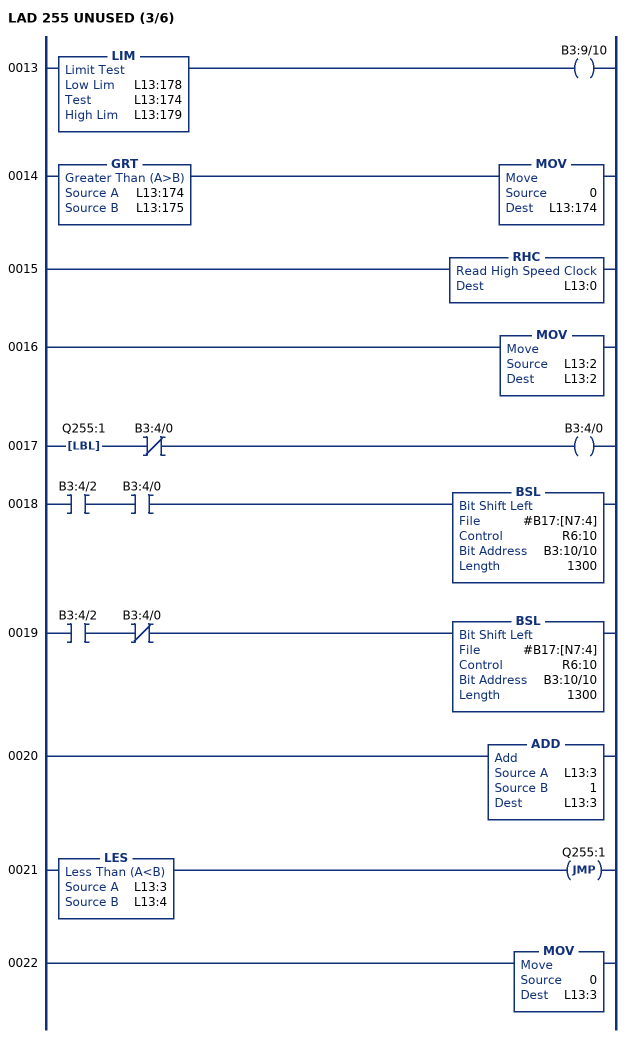
% Rung: 13 %
SOR LIM L13:178 L13:174 L13:179 OTE B3:9/10 EOR
% Rung: 14 %
SOR GRT L13:174 L13:175 MOV 0 L13:174 EOR
% Rung: 15 %
SOR RHC L13:0 EOR
% Rung: 16 %
SOR MOV L13:2 L13:2 EOR
% Rung: 17 %
SOR LBL Q255:1 XIO B3:4/0 OTE B3:4/0 EOR
% Rung: 18 %
SOR XIC B3:4/2 XIC B3:4/0 BSL #B17:[N7:4] R6:10 B3:10/10 1300 EOR
% Rung: 19 %
SOR XIC B3:4/2 XIO B3:4/0 BSL #B17:[N7:4] R6:10 B3:10/10 1300 EOR
% Rung: 20 %
SOR ADD L13:3 1 L13:3 EOR
% Rung: 21 %
SOR LES L13:3 L13:4 JMP Q255:1 EOR
% Rung: 22 %
SOR MOV 0 L13:3 EOR

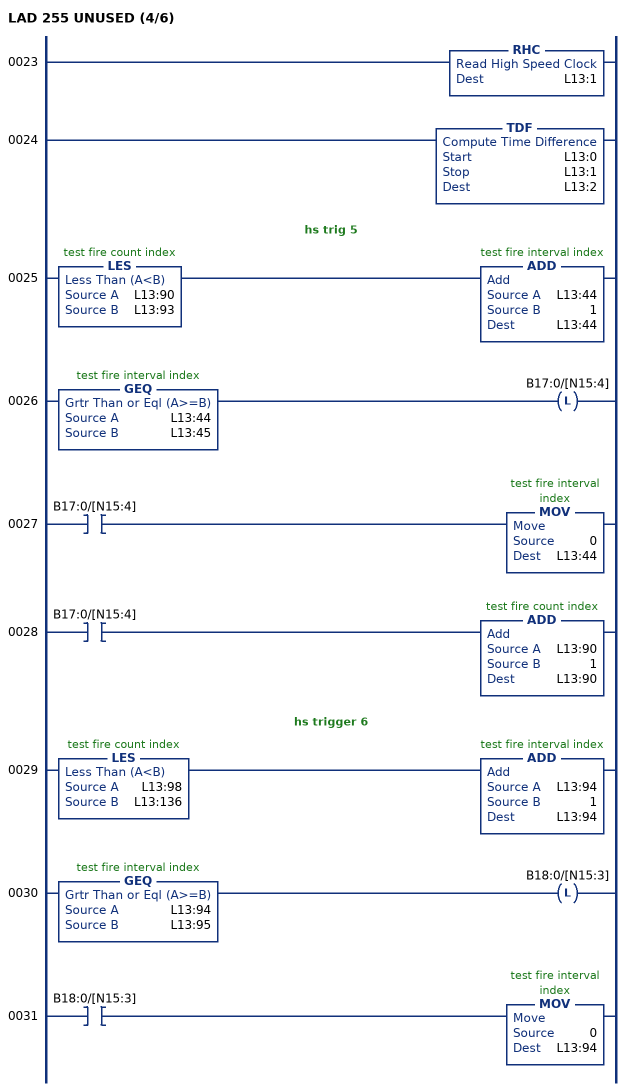
% Rung: 23 %
SOR RHC L13:1 EOR
% Rung: 24 %
SOR TDF L13:0 L13:1 L13:2 EOR
% Rung: 25 %
% TITLE: hs trig 5 %
SOR LES L13:90 L13:93 ADD L13:44 1 L13:44 EOR
%   L13:90  "test fire count index" %
%   L13:93  "test fire count" %
%   L13:44  "test fire interval index" %
% Rung: 26 %
SOR GEQ L13:44 L13:45 OTL B17:0/[N15:4] EOR
%   L13:44  "test fire interval index" %
%   L13:45  "test fire interval" %
%   B17:0  GOOD1 %
%   N15:4  INS_5_TRIG_LOC %
% Rung: 27 %
SOR XIC B17:0/[N15:4] MOV 0 L13:44 EOR
%   B17:0  GOOD1 %
%   N15:4  INS_5_TRIG_LOC %
%   L13:44  "test fire interval index" %
% Rung: 28 %
SOR XIC B17:0/[N15:4] ADD L13:90 1 L13:90 EOR
%   B17:0  GOOD1 %
%   N15:4  INS_5_TRIG_LOC %
%   L13:90  "test fire count index" %
% Rung: 29 %
% TITLE: hs trigger 6 %
SOR LES L13:98 L13:136 ADD L13:94 1 L13:94 EOR
%   L13:98  "test fire count index" %
%   L13:136  "test fire count" %
%   L13:94  "test fire interval index" %
% Rung: 30 %
SOR GEQ L13:94 L13:95 OTL B18:0/[N15:3] EOR
%   L13:94  "test fire interval index" %
%   L13:95  "test fire interval" %
%   B18:0  GOOD2 %
%   N15:3  INS_6_TRIG_LOC %
% Rung: 31 %
SOR XIC B18:0/[N15:3] MOV 0 L13:94 EOR
%   B18:0  GOOD2 %
%   N15:3  INS_6_TRIG_LOC %
%   L13:94  "test fire interval index" %

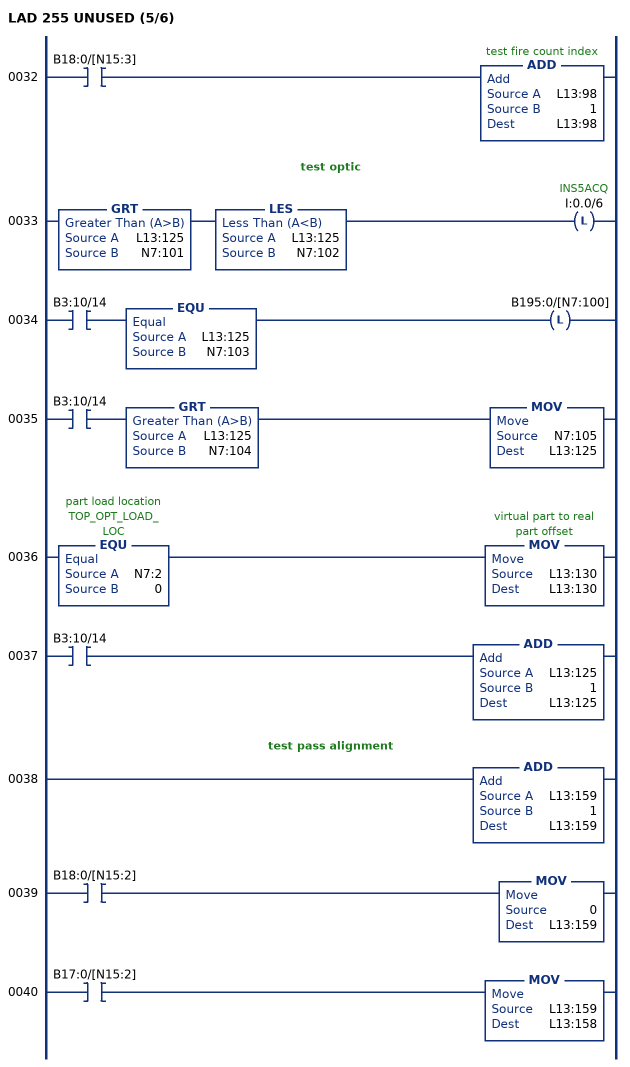
% Rung: 32 %
SOR XIC B18:0/[N15:3] ADD L13:98 1 L13:98 EOR
%   B18:0  GOOD2 %
%   N15:3  INS_6_TRIG_LOC %
%   L13:98  "test fire count index" %
% Rung: 33 %
% TITLE: test optic %
SOR GRT L13:125 N7:101 LES L13:125 N7:102 OTL I:0.0/6 EOR
%   I:0.0/6  INS5ACQ %
% Rung: 34 %
SOR XIC B3:10/14 EQU L13:125 N7:103 OTL B195:0/[N7:100] EOR
%   B195:0  TOP_NG %
% Rung: 35 %
SOR XIC B3:10/14 GRT L13:125 N7:104 MOV N7:105 L13:125 EOR
% Rung: 36 %
SOR EQU N7:2 0 MOV L13:130 L13:130 EOR
%   N7:2  TOP_OPT_LOAD_LOC  "part load location" %
%   L13:130  "virtual part to real part offset" %
% Rung: 37 %
SOR XIC B3:10/14 ADD L13:125 1 L13:125 EOR
% Rung: 38 %
% TITLE: test pass alignment %
SOR ADD L13:159 1 L13:159 EOR
% Rung: 39 %
SOR XIC B18:0/[N15:2] MOV 0 L13:159 EOR
%   B18:0  GOOD2 %
%   N15:2  BLOW_PT %
% Rung: 40 %
SOR XIC B17:0/[N15:2] MOV L13:159 L13:158 EOR
%   B17:0  GOOD1 %
%   N15:2  BLOW_PT %

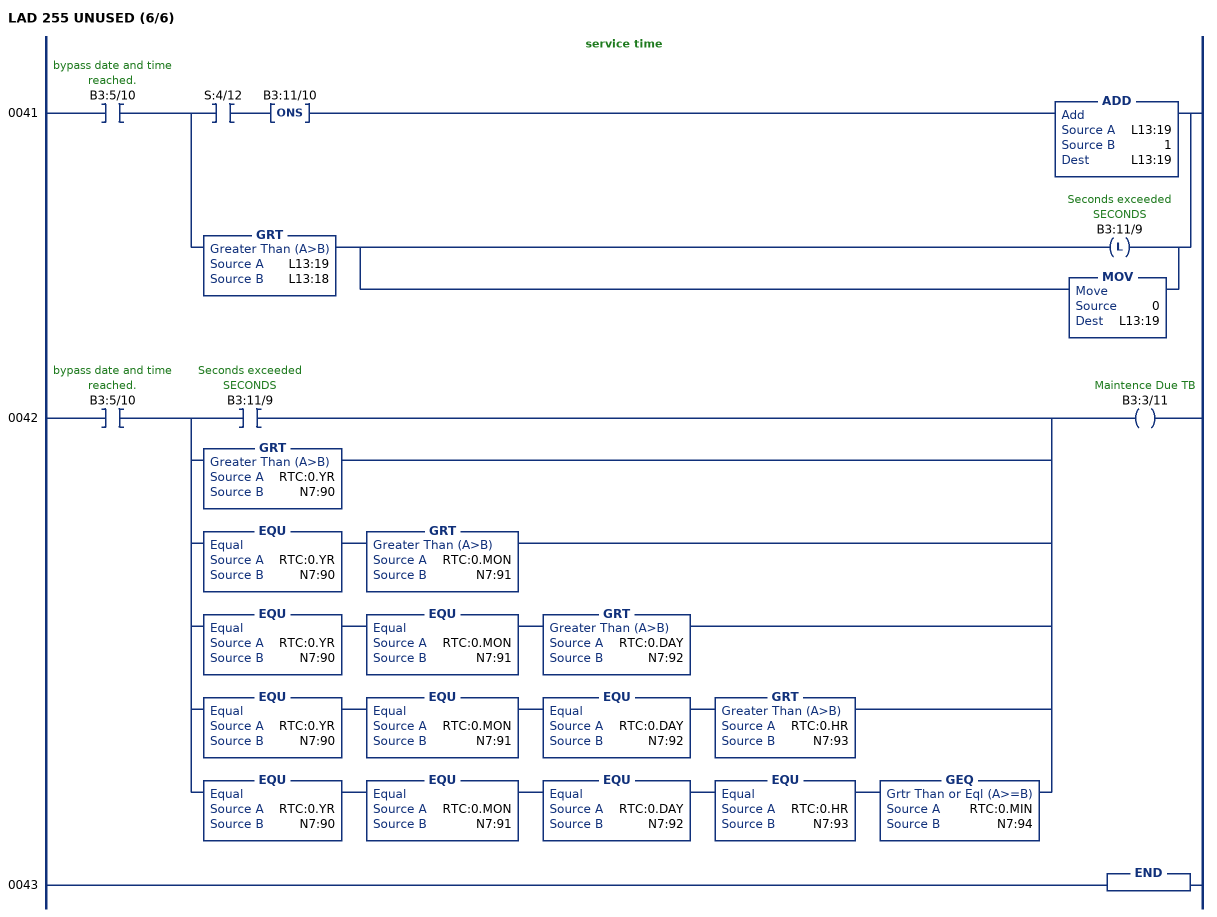
% Rung: 41 %
% TITLE: service time %
SOR XIC B3:5/10 BST XIC S:4/12 ONS B3:11/10 ADD L13:19 1 L13:19 NXB GRT L13:19 L13:18 BST OTL B3:11/9 NXB MOV 0 L13:19 BND BND EOR
%   B3:5/10  "bypass date and time reached." %
%   L13:18  MAX %
%   B3:11/9  SECONDS  "Seconds exceeded" %
% Rung: 42 %
SOR XIC B3:5/10 BST XIC B3:11/9 NXB GRT RTC:0.YR N7:90 NXB EQU RTC:0.YR N7:90 GRT RTC:0.MON N7:91 NXB EQU RTC:0.YR N7:90 EQU RTC:0.MON N7:91 GRT RTC:0.DAY N7:92 NXB EQU RTC:0.YR N7:90 EQU RTC:0.MON N7:91 EQU RTC:0.DAY N7:92 GRT RTC:0.HR N7:93 NXB EQU RTC:0.YR N7:90 EQU RTC:0.MON N7:91 EQU RTC:0.DAY N7:92 EQU RTC:0.HR N7:93 GEQ RTC:0.MIN N7:94 BND OTE B3:3/11 EOR
%   B3:5/10  "bypass date and time reached." %
%   B3:11/9  SECONDS  "Seconds exceeded" %
%   N7:90  RTC %
%   B3:3/11  TB  "Maintence Due" %
% Rung: 43 %
SOR END EOR

OTHER DOCUMENTED ADDRESSES
  B3  
  B196:0/2  ON
  B196:0/3  OFF
  B196:0/10  TOP_MOVE  "top movement detected"
  B196:1/2  DOWNTRACK_OPTIC_RUN  "Feed Bowl optic Run Signal after timing delays"
  I:0.0/0  TOP_CONV_ENC_A
  I:0.0/1  TOP_CONV_ENC_B
  I:0.0/8  INS5NG
  I:0.7  "Air Presure Sensor Input Signal"
  L42:0/2  "box full read (unused)"
  L42:1/1  "ps stop write (unused)"
  L199:9  "ones"
  L199:10  "billions"
  N15:9  FEED_WHEEL_STOP_TIME
  N197:7  "down track on delay"
  N197:8  "down track off delay"
  O:0.0/0  "spare"
  O:0.0/9  "spare"
  O:0.0/10  "spare"
  O:0.0/11  "spare"
  PFILE:6  "check for part jams"
  PFILE:10  "Bottom belt HSC"
  PFILE:12  "Top belt HSC"
  Q2:55  END_OF_MAIN
  U:6  "feed"
  U:217  "test trigger"

COMMENTS NOT ATTACHED TO A CURRENT RUNG
  F8:13: *************************
    Loads Side Camera Passing data into a bit shift
    *************************
    
    loads passing data bit into passing data bit shift register at the part present cl.
  I:0.0/8: special rung for testing. This rung can simulate a pass signal. It will not be timed correctly.
  B23:0/0: Yet another bit shift load with data in the part position indicating that there was a bottom system part pass as well as a top system part present at this location.
    
    verified works w/bypassed 071910 and unbypassed 072010
  C5:4: tempory counting to verify pass part count with boxing part count.
  B22:0/0: ***********************
     Bottom Part Syncronizing Logic
    ***********************
    
    This is the point at the bottom of the top conveyor where the part jumps from the bottom conveyor.  This system will then track the part through the top system to the point of the laser optic in order to verify that the part in question has passed the bottom inspection.  I believe that we NEED to include FAILING inspections to eliminate the possibility of a out of position part from passing. LW 072010
  T20:2.ACC: This rung is starting a timer that should be activated directly before the laser optic part presense sensor on the top conveyer and should cause the top optic to be ignored if the bottom camera system didn't pass. however other arrangements must be made if the bottom camera isn't going to be used as is the case with a nut inspection.
  T20:2: The timer used to verify that the part that triggered the top laser optic has passed the bottom camer. needs to be count
  N17:8: ****************************************************************************************************************
    I can not find anywhere in the program where the "Test Spacing From Pickup to Trigger is activated indicating to me that this entire function must not be doing anything in this program at this time.
    ****************************************************************************************************************
  B11:0/0: load part present bit shit with one shot data from the part present sensor
  B3:7/9: ************************************
     The next 3 rungs appear to do nothing
    ***********************************
  B9:0/[N7:47]: Remove any part present signals outside of expected location
  B9:0/[N7:50]: Remove any part present signals outside of expected location
  F19:0: Counter inside of a high speed counter interrupt counts the number of Bit Shifts that need to be processed in order to move the logic with the parts on the conveyor.
  F8:14: **************
    Bottom Top Camera Trigger
    *************
    
    Trigger Bottom Top Camera
  N10:4: test if boxing is connected
  B3:11/3: After initial delay allow blow two start functioning
  RUNG000150-000011: trigger count
  RUNG000150-000012: wipe stored part data if acq time expires
  RUNG000150-000013: clear data for aquire time expired
  RUNG000150-000014: clear data for time
  RUNG000150-000016: wiped count
  RUNG000150-000018: pass, fail and acquire inputs
  RUNG000150-000025: pass code / Set pass bit in Bit Shift
    captures result position and processing time
    Unlatch pass bit
  RUNG000150-000032: pass count
  RUNG000150-000035: fail count
  RUNG000150-000038: acquire code
  RUNG000150-000039: Grab trigger/acquire position
    Grab acquire time
  RUNG000150-000041: transfer tracked part positon from trigger/acquire to the acquire/result
    capture acquire time
    reset process time
  L14:8: on when ok for run
  L14:3: off when ok to run
  L14:2: off when ok to run
  L14:5: on when ok to run, rear off turns both off
  L13:165: maximum q i1
  N7:76: removed relieance on trigger signal
  N197:20/0: Passes deformed head blowoff command to TOP PLC where solenoid output is located.
  L13:162: maximum q
  L13:163: maximum average q
  B3:10/1: prevents momentary signals from box present sensor from tripping the logic for box not present
    
    This is in responce to a problem created by the sensor occasionally turning on as if no box was in its path when there is a box present.
  B3:6/2: IF PROCESSING FAULT OCURES AT COUNTER SENSOR; CLEAR THE BELT OF PASSING DATA
  L14:23: ****************  nEEDS fIXING  **********************
  L14:36: ****************  nEEDS fIXING  **********************
  RUNG000010-000014: ****
                      Zeros out the non passing part count when one passes
    ****
  RUNG000010-000018: Remove any part present signals outside of expected location
  T4:26: Check for buffer reset
  RUNG000125-000014: clear data for time
  RUNG000125-000013: clear data for aquire time expired
  RUNG000125-000012: wipe stored part data if acq time expires
  RUNG000125-000011: trigger count
  RUNG000125-000029: Set pass bit in Bit Shift
    captures result position and processing time
    Unlatch pass bit
  RUNG000125-000027: transfer tracked part positon from trigger/acquire to the acquire/result
    capture acquire time
    reset process time
  RUNG000125-000026: Grab trigger/acquire position
    Grab acquire time
  RUNG000125-000025: pass code / Set pass bit in Bit Shift
    captures result position and processing time
    Unlatch pass bit
  RUNG000125-000018: pass, fail and acquire inputs
  RUNG000125-000016: wiped count

REVISION NOTES
  13: updated count reset
  14: added io moduals
  15: multiple steps toward new hmi integration
  21: test

DATA TABLE (non-zero values as saved)
DATA B3
% B3:0 % 0X0120 0X0060 0X02C9 0XA000 0XA92E 0X2061 0X08A2 0X2AA6 0X2130 0X6104
% B3:10 % 0X8082 0X084C 0X2000 0X0000 0X0000 0X0000 0X0000 0X0000 0X0000 0X0000
DATA T4
% .PRE .ACC %
% T4:0 % 555 468
% T4:1 % 222 21
% T4:2 % 600 0
% T4:3 % 1000 1000
% T4:4 % 1 0
% T4:5 % 666 0
% T4:6 % 30 0
% T4:7 % 250 0
% T4:8 % 250 0
% T4:9 % 50 24
% T4:10 % 200 200
% T4:11 % 666 0
% T4:12 % 40 80
% T4:13 % 6 3
% T4:14 % 250 0
% T4:15 % 222 119
% T4:16 % 222 122
% T4:17 % 100 75
% T4:18 % 30 0
% T4:19 % 300 0
% T4:20 % 200 0
% T4:21 % 200 0
% T4:22 % 200 0
% T4:23 % 250 0
% T4:24 % 100 0
% T4:25 % 100 0
% T4:26 % 10 11
% T4:27 % 21 0
% T4:28 % 250 0
% T4:29 % 5000 0
% T4:30 % 50 50
% T4:31 % 20 0
% T4:32 % 69 0
DATA C5
% .PRE .ACC %
% C5:0 % 32766 0
DATA R6
% .LEN .POS %
% R6:0 % 2048 0
% R6:1 % 2048 0
% R6:2 % 3 0
% R6:3 % 3 0
% R6:4 % 1250 0
% R6:5 % 1250 0
% R6:6 % 1250 0
% R6:7 % 10 0
% R6:8 % 3 0
% R6:9 % 3 0
% R6:10 % 1300 0
% R6:11 % 1300 0
% R6:12 % 10 0
% R6:13 % 10 0
% R6:14 % 10 0
% R6:15 % 10 0
% R6:16 % 1100 0
% R6:17 % 1440 0
% R6:18 % 1440 0
% R6:19 % 10 0
DATA N7
% N7:0 % 3339 1 1168 0 0 0 49 0 1 0
% N7:10 % 48 62 1 47 1378 250 555 100 32468 96
% N7:20 % 0 73 0 0 1 10 9 1190 4096 13
% N7:30 % 50 9 800 555 222 3 1533 222 1165 222
% N7:40 % 2100 2158 10 5 2153 10 101 2050 50 1542
% N7:50 % 1552 800 10 41 0 0 1542 1552 10 41
% N7:60 % 0 0 1051 40 47 1946 1947 1944 1943 0
% N7:70 % 0 21 23 27738 32767 0 122 0 16 0
% N7:80 % 0 6 95 0 0 0 5 500 0 0
% N7:90 % 2011 4 4 12 1 0 0 0 0 1600
% N7:100 % 1003 90 110 100 175 25 0 0 0 0
DATA F8
% F8:0 % 18 206.64 23807 499 0.23807
% F8:5 % 0 0 500 1.9 2
% F8:10 % 1 0.08897486 0 101 63.26563
% F8:15 % 37.73437 4040 2 0 0
% F8:20 % 0 0.02 0 1 0
% F8:25 % 0 932781 0.222 279.6551 848597
% F8:30 % 0 170 0.03 38 852060
% F8:35 % 0 0 0 0 77
% F8:40 % 101 37.73437 0 100 1
% F8:45 % 1 2 0.21455 0 0
% F8:50 % 0 0 1 0 1
% F8:55 % 2000000 -221 0 0 0
% F8:95 % 0 0 0 492 4.92
DATA B12
% B12:0 % 0X0554 0X0000 0X0000 0X0000 0X0000 0X0000 0X0000 0X0000 0X0000 0X0000
DATA L13
% L13:0 % 308402300 308407124 4824 0 1000
% L13:5 % 0 -1901611778 100 1162124017 1162124017
% L13:10 % 492 300 78447 0 -885760695
% L13:15 % -1282263690 -2147483648 2147483647 2147483647 82058
% L13:20 % 6000000 -1295363090 0 -1144258314 2035272617
% L13:25 % 27 849 623 0 1000000000
% L13:30 % -1144259014 78452 2044398469 13 156899
% L13:35 % 678 156899 2044398469 37 2035272617
% L13:40 % -1283018330 0 19 20 0
% L13:45 % 60 700 27 0 16
% L13:50 % 0 35 666 50 3
% L13:55 % 0 1353 1297 226 226
% L13:60 % 8 10576 13 2044398343 12
% L13:65 % 650492 20 379089 1507595048 5501
% L13:70 % 1507612018 1507611965 53 0 5500
% L13:75 % -1 10 2377213 -1313930933 2377
% L13:80 % 27 -47 18250 0 999999
% L13:85 % 6475 291 44441 -1282752161 -1282751687
% L13:90 % 26616 0 0 1000 0
% L13:95 % 60 0 0 25989 488545
% L13:100 % 488093 -1282752128 -1282751656 4 3
% L13:105 % -1295599743 -1295599743 0 0 0
% L13:110 % 75 33 31 -1303967890 -1303588810
% L13:115 % -1303588792 18 9 -1303588801 5
% L13:120 % 33 10337 19 30 31
% L13:125 % 164 -1295599743 -1295599743 13 13
% L13:130 % 5 0 1 558 0
% L13:135 % 0 1000 226 12 0
% L13:140 % 0 1 12 0 20
% L13:145 % 1 34396982 35155 6 6
% L13:150 % 5 5 5 5 5
% L13:155 % 5 5 24 0 168160
% L13:160 % 3 5 4 395082 53203921
% L13:165 % 3 189116 95 13 0
% L13:170 % 55946610 0 0 1 30
% L13:175 % 300 5 5 0 10
% L13:180 % 5 6946 1000 22 1000
% L13:185 % 55 172460 60 1 720323
% L13:190 % 65 0 1 379089 379089
% L13:195 % -2370948 2370948 0 0 0
DATA F14
% F14:0 % 760.1599 200.1099 76 20 15
% F14:5 % 32766 21297.9 0 0 0
DATA N15
% N15:0 % 100 889 1945 1201 1200 134 105 100 1159 10
% N15:10 % 61 504 0 0 0 0 1172 0 0 0
DATA L16
% L16:0 % 12 40 72 0 20
% L16:5 % 250 5000 5000 182 19
% L16:10 % 1256 18 2045 6599584 98
% L16:15 % 99 0 0 0 0
DATA B17
% B17:50 % 0X0000 0X0010 0X0000 0X0000 0X0000 0X0000 0X0000 0X0000 0X0000 0X0000
DATA B18
% B18:50 % 0X0000 0X0010 0X0000 0X0000 0X0000 0X0000 0X0000 0X0000 0X0000 0X0000
% B18:60 % 0XC000 0X0000 0X0000 0X0000 0X0000 0X0000 0X0000 0X0000 0X0000 0X0000
DATA L19
% L19:0 % -1144266694 -1144265339 -1144265113 -1144263756 -1144263531
% L19:5 % -1144262174 -1144261949 -1144260596 -1144260370 -1144259014
% L19:10 % -1144258788 -1144296955 -1144296727 -1144295373 -1144295147
% L19:15 % -1144293793 -1144293568 -1144292213 -1144291988 -1144290632
% L19:20 % -1144290404 -1144289051 -1144288825 -1144287470 -1144287244
% L19:25 % -1144285888 -1144285664 -1144284312 -1144284086 -1144282731
% L19:30 % -1144282504 -1144281152 -1144280926 -1144279570 -1144279344
% L19:35 % -1144277988 -1144277763 -1144276410 -1144276184 -1144274826
% L19:40 % -1144274600 -1144273248 -1144273021 -1144271667 -1144271441
% L19:45 % -1144270087 -1144269861 -1144268503 -1144268276 -1144266921
DATA L20
% L20:0 % 2072136995 2072136995 2072136995 2072136995 2072136995
% L20:5 % 2072136995 2072136995 2072136995 2072136995 2072136995
% L20:10 % 2072136995 2072136995 2072136995 2072136995 2072136995
% L20:15 % 2072136995 2072136995 2072136995 2072136995 2072136995
% L20:20 % 2072136995 2072136995 2072136995 2072136995 2072136995
% L20:25 % 2072136995 2072136995 2072136995 2072136995 2072136995
% L20:30 % 2072136995 2072136995 2072136995 2072136995 2072136995
% L20:35 % 2072136995 2072136995 2072136995 2072136995 2072136995
% L20:40 % 2072136995 2072136995 2072136995 2072136995 2072136995
% L20:45 % 2072136995 2072136995 2072136995 2072136995 2072136995
DATA L21
% L21:0 % -1144296045 -1144294690 -1144294463 -1144293109 -1144292883
% L21:5 % -1144291527 -1144291301 -1144289948 -1144289722 -1144288365
% L21:10 % -1144288138 -1144286784 -1144286558 -1144285206 -1144284981
% L21:15 % -1144283624 -1144283398 -1144282042 -1144281817 -1144280464
% L21:20 % -1144280238 -1144278886 -1144278660 -1144277303 -1144277076
% L21:25 % -1144275718 -1144275492 -1144274137 -1144273911 -1144272559
% L21:30 % -1144272332 -1144270977 -1144270750 -1144269393 -1144269167
% L21:35 % -1144267809 -1144267584 -1144266229 -1144266003 -1144264646
% L21:40 % -1144264419 -1144263062 -1144262836 -1144261481 -1144261254
% L21:45 % -1144259899 -1144259674 -1144258314 -1144258088 -1144296272
DATA L22
% L22:0 % 2072136995 2072136995 2072136995 2072136995 2072136995
% L22:5 % 2072136995 2072136995 2072137059 2072136995 2072136995
% L22:10 % -75280985 2072136995 2072137067 2072137059 2072137523
% L22:15 % 2072137059 2072137059 2072136995 2072137059 2072136995
% L22:20 % 2072136995 -74821853 2072136995 2139245859 2072136995
% L22:25 % 2072136995 2072145779 2074242403 2073189795 -75346653
% L22:30 % 2072399203 2072136995 2072136995 2072136995 2072407459
% L22:35 % 2072669475 2072136995 2072136995 2072136995 2072136995
% L22:40 % 2072169831 2141343523 2072136995 2072136995 2074234147
% L22:45 % 2072169891 2074496803 2072247603 2074234147 2072136995
DATA L23
% L23:0 % -1304697501 -1304696943 -1304696384 -1304695825 -1304695268
% L23:5 % -1304694711 -1304694153 -1282753837 -1282753278 -1282752719
% L23:10 % -1282752161 -1304719281 -1304718723 -1304718164 -1304717606
% L23:15 % -1304717048 -1304716490 -1304715930 -1304715371 -1304714813
% L23:20 % -1304714254 -1304713694 -1304713136 -1304712578 -1304712020
% L23:25 % -1304711462 -1304710903 -1304710345 -1304709788 -1304709228
% L23:30 % -1304708671 -1304708112 -1304707554 -1304706995 -1304706437
% L23:35 % -1304705879 -1304705321 -1304704763 -1304704205 -1304703647
% L23:40 % -1304703088 -1304702530 -1304701970 -1304701411 -1304700853
% L23:45 % -1304700292 -1304699733 -1304699175 -1304698617 -1304698059
DATA L24
% L24:0 % -1295599743 -1295599743 -1295599743 -1295599743 -1295599743
% L24:5 % -1295599743 -1295599743 -1295599743 -1295599743 -1295599743
% L24:10 % -1295599743 -1295599743 -1295599743 -1295599743 -1295599743
% L24:15 % -1295599743 -1295599743 -1295599743 -1295599743 -1295599743
% L24:20 % -1295599743 -1295599743 -1295599743 -1295599743 -1295599743
% L24:25 % -1295599743 -1295599743 -1295599743 -1295599743 -1295599743
% L24:30 % -1295599743 -1295599743 -1295599743 -1295599743 -1295599743
% L24:35 % -1295599743 -1295599743 -1295599743 -1295599743 -1295599743
% L24:40 % -1295599743 -1295599743 -1295599743 -1295599743 -1295599743
% L24:45 % -1295599743 -1295599743 -1295599743 -1295599743 -1295599743
DATA L25
% L25:0 % -1282767881 -1282767655 -1282767430 -1282767205 -1282766980
% L25:5 % -1282766755 -1282766529 -1282766305 -1282766079 -1282765855
% L25:10 % -1282765628 -1282765402 -1282765177 -1282764951 -1282764727
% L25:15 % -1282764501 -1282764276 -1282764050 -1282763825 -1282763600
% L25:20 % -1282756416 -1282756192 -1282755967 -1282755743 -1282755517
% L25:25 % -1282755291 -1282755067 -1282754841 -1282754616 -1282754391
% L25:30 % -1282754165 -1282753940 -1282753715 -1282753489 -1282753264
% L25:35 % -1282753038 -1282752813 -1282752589 -1282752362 -1282752137
% L25:40 % -1282751913 -1282751687 -1282769681 -1282769457 -1282769231
% L25:45 % -1282769006 -1282768781 -1282768556 -1282768330 -1282768106
DATA L26
% L26:0 % -1295599743 -1295599743 -1295599743 -1295599743 -1295599743
% L26:5 % -1295599743 -1295599743 -1295599743 -1295599743 -1295599743
% L26:10 % -1295599743 -1295599743 -1295599743 -1295599743 -1295599743
% L26:15 % -1295599743 -1295599743 -1295599743 -1295599743 -1295599743
% L26:20 % -1295599743 -1295599743 -1295599743 -1295599743 -1295599743
% L26:25 % -1295599743 -1295599743 -1295599743 -1295599743 -1295599743
% L26:30 % -1295599743 -1295599743 -1295599743 -1295599743 -1295599743
% L26:35 % -1295599743 -1295599743 -1295599743 -1295599743 -1295599743
% L26:40 % -1295599743 -1295599743 -1295599743 -1295599743 -1295599743
% L26:45 % -1295599743 -1295599743 -1295599743 -1295599743 -1295599743
DATA L27
% L27:0 % -1901611778 -1053149009 -1053120077 -1053089810 -1053059766
% L27:5 % -1053030628 -1053001435 -1052971494 -1052940423 -1052879062
% L27:10 % -1052848887 -1052818882 -1052787634 -1052754762 -1052712702
% L27:15 % -1052672799 -1052630656 -1052597913 -1052564740 -1052530450
% L27:20 % -1052497221 -1051786034 -1054274552 -1054246135 -1054212963
% L27:25 % -1054174819 -1054143079 -1054112165 -1054080515 -1054044002
% L27:30 % -1054002897 -1053968417 -1053936847 -1053891811 -1053839091
% L27:35 % -1053804013 -1053767217 -1053733357 -1053540607 -1053506211
% L27:40 % -1053473370 -1053445569 -1053414718 -1053383869 -1053353708
% L27:45 % -1053325991 -1053297789 -1053269322 -1053239598 -1053210393
DATA L42
% L42:0 % -734706044 -2042345216 570425412 67108864 1075986433
% L42:5 % 262191 276824237 9519149 12864 1024
% L42:10 % 143654912 8466 -2147467264 281088 0
% L42:15 % 4672 16384 -2080374784 134217728 268435456
% L42:20 % 32776 1048580 33587198 536903678 16384
% L42:25 % 1408 524288 8388608 572522752 38019072
% L42:30 % 0 68161536 807422080 84 0
% L42:35 % 71565376 69888 537411584 0 256
% L42:40 % 0 272 67108864 138936320 37752833
% L42:45 % 1053696 32784 1048576 131072 4160
% L42:50 % 536870912 542
DATA B181
% B181:0 % 0X0040 0X0040 0X0000 0X0000 0X0800 0X0000 0X0010 0X2004 0X0000 0X0001
% B181:10 % 0X0004 0X0000 0X0002 0X3000 0X0000 0X0000 0X0000 0X0001 0X0000 0X0080
% B181:20 % 0X0000 0X0000 0X8004 0X1000 0X8000 0X0000 0X0000 0X0002 0X0000 0X0000
% B181:30 % 0X0000 0X0020 0X0000 0X1000 0X0004 0X6080 0X0000 0X0004 0X0002 0X0000
% B181:40 % 0X0000 0X8020 0X0044 0X0018 0X0040 0X2800 0X0500 0X4020 0X0080 0X2000
% B181:50 % 0X0000 0X0000 0X8000 0X0040 0X0000 0X0002 0X0000 0X0000 0X0000 0X0000
% B181:60 % 0X0400 0X1140 0X0000 0X0000 0X0000 0X0000 0X0000 0X0000 0X0000 0X0040
% B181:70 % 0X0100 0X0000 0X0000 0X0000 0X60C1 0X0200 0X0200 0X1010 0X0000 0X0000
% B181:80 % 0X0008 0X0000 0X8001 0X2200 0X00A0 0X0004 0X2000 0X0000 0X0100 0X0450
% B181:90 % 0X0001 0X0A00 0X0800 0X0001 0X0010 0X0200 0X1200 0X0004 0X0042 0X0020
% B181:100 % 0X0000 0X0000 0X0000 0X4000 0X8000 0X0000 0X0000 0X0000 0X0080 0X0001
% B181:110 % 0X4200 0X0000 0X0000 0X0000 0X8000 0X0000 0X0000 0X0004 0X0008 0X4000
% B181:120 % 0X0200 0X0028 0X0000 0X0401 0X1080 0X0100 0X8001 0X0000 0X0100 0X0402
% B181:130 % 0X0020 0X0000 0X0010 0X8002 0X0000 0X8000 0X0008 0X0120 0X0000 0X0000
% B181:140 % 0X0000 0X0002 0X0110 0X0000 0X0010 0X0000 0X1040 0X0000 0X0104 0X0000
% B181:150 % 0X0000 0X0000 0X1910 0X9800 0X0008 0X4600 0X0004 0X0111 0X0002 0X0000
% B181:160 % 0X0000 0X0000 0X4222 0X8B22 0X0000 0X2000 0XC880 0X2044 0X0042 0X0100
% B181:170 % 0XC808 0X0098 0X4089 0X0048 0X0091 0X1120 0X4580 0X008A 0X0000 0X0910
% B181:180 % 0X0000 0X8001 0X0048 0X0244 0X1800 0X8088 0X0080 0X0010 0X8000 0X4000
% B181:190 % 0X0044 0X1800 0X0245 0X0000 0X0000 0X0000 0X0000 0X0000 0X0000 0X0000
% B181:200 % 0X0000 0X1008 0X0011 0X0000 0X4880 0X0100 0X0082 0X4000 0X0000 0X0000
% B181:210 % 0X4004 0X2000 0X1011 0X0028 0X0444 0X8000 0X0000 0X0000 0X0000 0X0800
% B181:220 % 0X3000 0X0000 0X0226 0X4002 0X0000 0X0000 0X2100 0X4540 0X0002 0X0200
% B181:230 % 0X0000 0X0002 0X1000 0X0000 0X0008 0X8040 0X0001 0X0000 0X1001 0X0012
% B181:240 % 0X0080 0X0000 0X0004 0X0000 0X0100 0X0000 0X0000 0X0400 0X2240 0X0800
% B181:250 % 0X0010 0X0000 0X0000 0X0020 0X0001 0X0000
DATA F182
% F182:0 % -7.703779e-34 2.529285e-29 7.174648e-43 0 2.295887e-41
% F182:5 % 5.739719e-42 3.587324e-43 2.938736e-39 262144 2.390736e-38
% F182:10 % 0 528 2.325539e-40 9.422322e-38 3.859385e-34
% F182:15 % 3.85186e-34 6.462349e-27 0 0 0
% F182:20 % 0 2.802597e-45 2.351132e-38 0 3.67342e-40
% F182:25 % 0 0 1.121039e-44 2.938915e-39 2.007812
% F182:30 % 7.34684e-40 9.18355e-41 0 3.67342e-40 8.96831e-44
% F182:35 % 2.938758e-39 5.739719e-42 7.174648e-43 -0 0
% F182:40 % 5.883211e-39 -2.000244 5.605194e-45 -2.524365e-29 0
% F182:45 % 2.602297e-18 1.084202e-19 2 9.404251e-38 0
DATA L183
% L183:0 % 1427522511 1968587600 1 -1147483520 536875040
% L183:5 % 321 262150 283 0 -2147483568
% L183:10 % 1074266112 134217856 2162688 570458112 8458244
% L183:15 % 4 2098176 0 1 1073741828
% L183:20 % 420483092 537921796 1024 152060992 134217728
% L183:25 % 1073741824 0 -2080357376 608174096 541065216
% L183:30 % 0 66048 516 33817600 524290
% L183:35 % 8945920 512 135274496 67117060 32
% L183:40 % 16777216 8388608 16384 32 2080
% L183:45 % 1224736768 287440900 8 42532864 -2139095040
DATA N184
% N184:0 % 8192 333 274 0 0 290 1024 0 64 2080
% N184:10 % 64 0 0 0 128 0 16384 136 513 2306
% N184:20 % 0 32 4 0 144 136 -32768 0 4096 4096
% N184:30 % 8194 0 4 0 0 1024 64 4 0 10368
% N184:40 % 68 0 2192 32 16896 68 0 0 0 2048
DATA B185
% B185:0 % 0X0202 0X0009 0X0000 0X0040 0X0200 0X1080 0X0040 0X0404 0X0020 0X0001
% B185:10 % 0X0100 0X0000 0X0801 0X0080 0X8000 0X0000 0X0800 0X0040 0X0040 0X0004
% B185:20 % 0X0040 0X0100 0X0010 0X0400 0X0040 0X0004 0X0400 0X0000 0XC280 0X2704
% B185:30 % 0X0042 0X0804 0X0000 0X0000 0X0102 0X0010 0X0201 0X0000 0X0100 0X8200
% B185:40 % 0X2000 0X0200 0X0110 0X0000 0X0000 0X0000 0X0091 0X0000 0X0000 0X0000
DATA N186
% N186:0 % 100 0 0 0 0 0 8256 16480 0 256
% N186:10 % 0 256 32 2048 2112 1176 0 8 1026 0
% N186:20 % 0 1 4608 0 256 16 0 16384 2 2560
% N186:30 % 0 0 0 -28672 132 2048 -32768 4 4608 1
% N186:40 % 128 0 -32224 128 128 0 32 16529 0 0
DATA L187
% L187:0 % 35913762 4194304 497 1073743907 50212
% L187:5 % 19495 0 0 67174428 544
% L187:10 % -2147418112 546312192 0 536870920 4096
% L187:15 % 67112960 0 4 268435456 33554432
% L187:20 % 67108864 135266368 1073881088 0 1091043328
% L187:25 % 268439552 128 16641 32768 1024
% L187:30 % 0 1073741888 8192 8192 0
% L187:35 % 4 -2147448704 1 0 32768
% L187:40 % 8650752 0 12582912 32776 402653184
% L187:45 % 553648128 67638 8192 262144 0
DATA F188
% F188:0 % 6.000977 66.00024 11 44.00001 29
% F188:5 % 0 0 -0 0 0
% F188:10 % 0 7.174648e-43 5.605194e-44 4.484155e-44 2.350989e-38
% F188:15 % 7.174648e-43 4.591775e-41 9.408547e-38 0 1.175499e-38
% F188:20 % 4.591775e-41 1.219727e-19 0 7.174648e-43 1.084467e-19
% F188:25 % 0 2.802597e-45 0 1.102026e-39 0
% F188:30 % 0 1.175495e-38 9.403955e-38 5.877472e-39 4.829871e-34
% F188:35 % 9.403955e-38 5.877472e-39 0 0 0
% F188:40 % 0 -7.34684e-40 3.85186e-34 1.528143e-36 0
% F188:45 % 0 4.484155e-44 6.018577e-36 1.793662e-43 9.550892e-38
DATA B189
% B189:0 % 0X20F0 0X0000 0X0040 0X0000 0X4104 0X0401 0X0000 0X0000 0X0000 0X0000
% B189:10 % 0X0000 0X1000 0X0082 0X0000 0X0000 0X0000 0X0001 0X0000 0X0000 0X0000
% B189:20 % 0X0040 0X0000 0X1000 0X0042 0X0001 0X0000 0X0000 0X0004 0X0000 0X0000
% B189:30 % 0X0000 0X0001 0X0000 0X0200 0X0C20 0X0001 0X0000 0X03B0 0X0008 0X0000
% B189:40 % 0X0000 0X0000 0X0015 0X0000 0X0000 0X0000 0X0000 0X011A 0X0000 0X0000
DATA L190
% L190:0 % 1 87 0 0 4198464
% L190:5 % 0 520 0 0 0
% L190:10 % 131072 65536 0 1 -2147483632
% L190:15 % 1082130432 0 512 1024 268435712
% L190:20 % 536870912 4 256 262400 0
% L190:25 % 32768 0 33570816 0 2097152
% L190:30 % 8667136 2 0 0 0
% L190:35 % 0 256 0 38912 0
% L190:40 % 0 131072 0 0 0
% L190:45 % 4194304 0 0 536903681 -2147481340
DATA B191
% B191:0 % 0X0008 0X0001 0X0000 0X8408 0X0000 0X0000 0X0000 0X0024 0X0040 0X8000
DATA L192
% L192:0 % -1444152502 266932201 5055 76 0
% L192:5 % 1000000 39200000 134220775 263143 72
% L192:10 % 1073872896 536870912 0 -1 -1
% L192:15 % 1507816393 -1 -1 100 0
% L192:20 % -1 279000000 -1 -1 -1
% L192:25 % -1 -1 -1 -1 -1
% L192:30 % -1 -1 -1 -1 -1
% L192:35 % -1 -1 -1 -1 -1
% L192:40 % -1 -1 -1 -1 -1
% L192:45 % -1 -1 -1 -1 -1
DATA B194
% B194:80 % 0X0100 0X0000 0X0000 0X1000 0X0000 0X0000 0X0100 0X0040 0X0000 0X4000
% B194:90 % 0X0000 0X0000 0X0000 0X0800 0X0000 0X0000 0X0000 0X0A10 0X0000 0X0880
% B194:100 % 0X0000 0X0000 0X0000 0X0008 0X0000 0X0000 0X0000 0X4000 0X0000 0X0100
% B194:110 % 0X0000 0X0000 0X0000 0X0000 0X0000 0X0008 0X0444 0X0000 0X0000 0X0000
% B194:120 % 0X0000 0X0000 0X0840 0X8000 0X0000 0X0080 0X0400 0X0000 0X2000 0X0000
% B194:130 % 0X0010 0X0004 0X0000 0X0000 0X0040 0X0080 0X0000 0X0004 0X0000 0X0080
% B194:140 % 0X0004 0X1000 0X0000 0X0000 0X0000 0X0001 0X0000 0X0000 0X0000 0X0000
% B194:150 % 0X0000 0X000C 0X2000 0X0000 0X0000 0X0000 0X0000 0X0000 0X0000 0X0000
% B194:160 % 0X0000 0X8000 0X0004 0X0000 0X0008 0X0000 0X0120 0X0010 0X0000 0X0002
% B194:170 % 0X0000 0X0000 0X0000 0X0000 0X0000 0X0040 0X0000 0X0000 0X0001 0X0000
% B194:180 % 0X0000 0X0400 0X0000 0X0000 0X0100 0X0000 0X0000 0X0440 0X0000 0X0010
% B194:190 % 0X2020 0X8000
